(* Schneider Machine Expert - Basic project control, file version 2.9.0.0 *)
(* ProjectInformations: Name=Nuevo proyecto *)

HARDWARE
  Cpu 0: TM221M16R/G
  EthernetConfiguration: NetworkName=M221, IpAllocationMode=FixedAddress, IpAddress=0.0.0.0, SubnetMask=0.0.0.0
  SerialLineConfiguration: Baud=Baud19200, Parity=ParityEven, DataBits=DataBits8, StopBits=StopBits1, PhysicalMedium=PhysicalMediumRs485, TransmissionMode=TransmissionModeModbusRtu, SlaveId=1, Addressing=SlaveAddressing
  MastTask: UsePeriodScanMode=true, PeriodScan=50
  FastTask: Period=255
  CpuBehavior: StartingMode=StartAsPreviousState, AutoSaveRamOnEeprom=true, WatchdogPeriod=250

SYMBOLS  (address, symbol, comment, settings)
  %MW103    CONT
  %MW500    POSITION
  %MW501    VELOCITY
  %MW502    ANGLE
  %MW503    CRISP
  %MF1      POS_NL
  %MF3      POS_NM
  %MF5      POS_NP
  %MF7      POS_ZR
  %MF9      POS_PP
  %MF11     POS_PM
  %MF13     POS_PL
  %MF15     VEL_NL
  %MF17     VEL_NM
  %MF19     VEL_NP
  %MF21     VEL_ZR
  %MF23     VEL_PP
  %MF25     VEL_PM
  %MF27     VEL_PL
  %MF29     ANG_NL
  %MF31     ANG_NM
  %MF33     ANG_ZR
  %MF35     ANG_PM
  %MF37     ANG_PL
  %MF39     W10
  %MF41     W23
  %MF43     W24
  %MF45     W2
  %MF47     W5
  %MF49     W11
  %MF51     W15
  %MF53     W18
  %MF55     W21
  %MF57     W22
  %MF59     W3
  %MF61     W6
  %MF63     W12
  %MF65     W17
  %MF67     W20
  %MF69     W1
  %MF71     W4
  %MF73     W7
  %MF75     W8
  %MF77     W13
  %MF79     W16
  %MF81     W19
  %MF83     W9
  %MF85     W14
  %MF87     W25
  %MF89     NL
  %MF91     NM
  %MF93     ZR
  %MF95     PM
  %MF97     PL
  %MF99     NUM
  %MF101    DEN
  %KF1      MEAN_NL_POS  [Value=-3]
  %KF3      MEAN_NM_POS  [Value=-2]
  %KF5      MEAN_NP_POS  [Value=-1]
  %KF7      MEAN_ZR_POS  [Value=0]
  %KF9      MEAN_PP_POS  [Value=1]
  %KF11     MEAN_PM_POS  [Value=2]
  %KF13     MEAN_PL_POS  [Value=3]
  %KF15     SIGMA_POS  [Value=0.365]
  %KF17     MEAN_NL_VEL  [Value=-5]
  %KF19     MEAN_NM_VEL  [Value=-3.333]
  %KF21     MEAN_NP_VEL  [Value=-1.667]
  %KF23     MEAN_ZR_VEL  [Value=0]
  %KF25     MEAN_PP_VEL  [Value=1.667]
  %KF27     MEAN_PM_VEL  [Value=3.333]
  %KF29     MEAN_PL_VEL  [Value=5]
  %KF31     SIGMA_VEL  [Value=0.7]
  %KF33     MEAN_NL_THETA  [Value=-0.2618]
  %KF35     MEAN_NM_THETA  [Value=-0.1]
  %KF37     MEAN_ZR_THETA  [Value=0]
  %KF39     MEAN_PM_THETA  [Value=0.1]
  %KF41     MEAN_PL_THETA  [Value=0.2618]
  %KF43     SIGMA_L_THETA  [Value=0.085]
  %KF45     SIGMA_M_THETA  [Value=0.03]
  %KF47     SIGMA_Z_THETA  [Value=0.02]
  %KF49     MEAN_U_NL  [Value=-200]
  %KF51     MEAN_U_NM  [Value=-100]
  %KF53     MEAN_U_ZR  [Value=0]
  %KF55     MEAN_U_PM  [Value=100]
  %KF57     MEAN_U_PL  [Value=200]
  %KF59     SIGMA_L_U  [Value=50]
  %KF61     SIGMA_M_U  [Value=45]
  %KF63     SIGMA_Z_U  [Value=35]

POU Fuzzy
  (* SectionNumber=1 *)

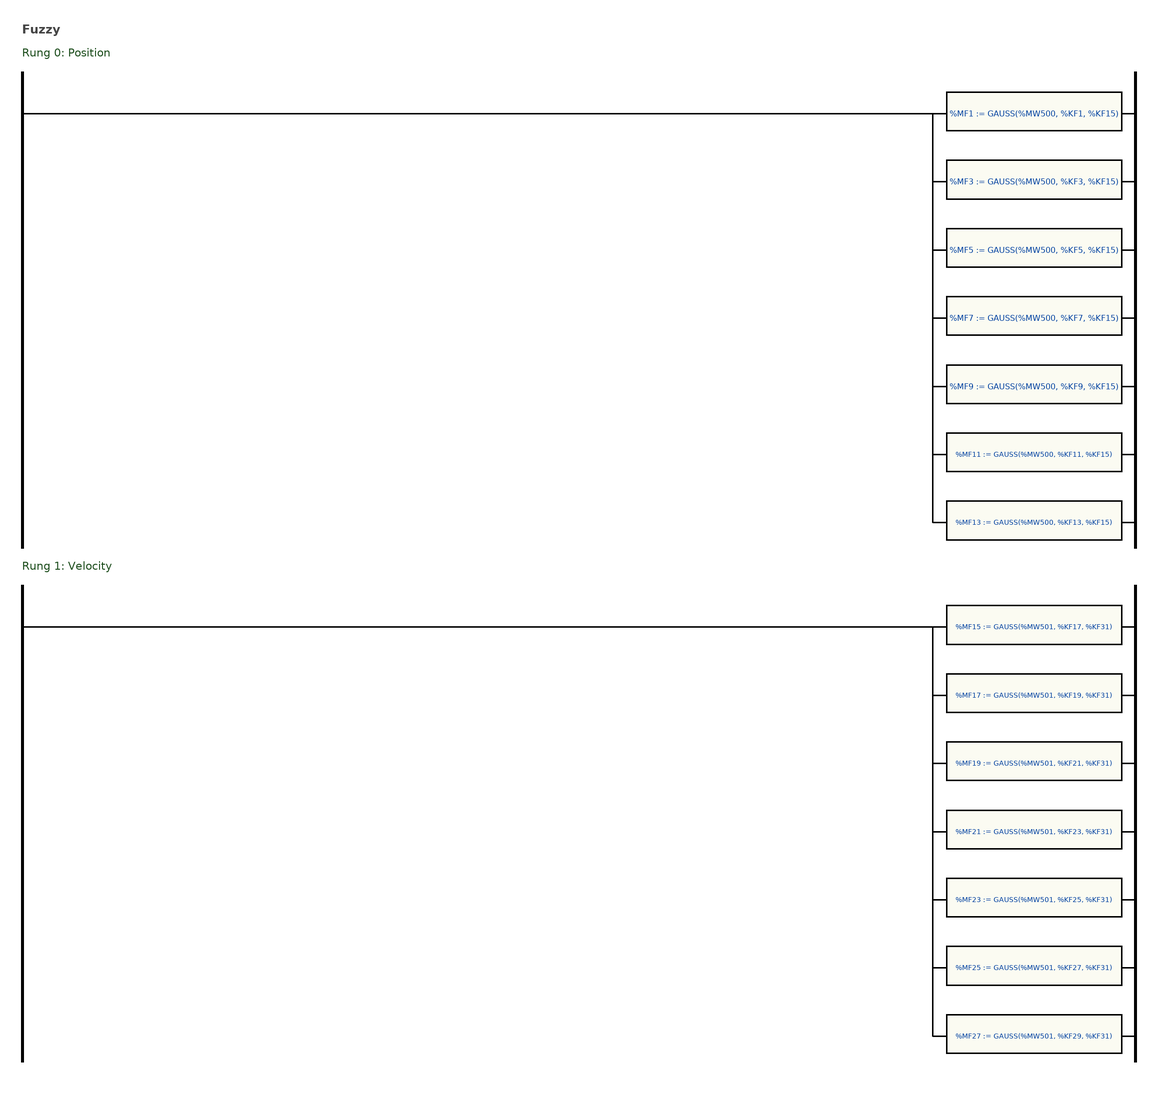

// Rung 0: Position
  LD 1
  [ %MF1 := GAUSS ( %MW500 , %KF1 , %KF15 ) ](* POS_NL, POSITION, MEAN_NL_POS, SIGMA_POS *)
  [ %MF3 := GAUSS ( %MW500 , %KF3 , %KF15 ) ](* POS_NM, POSITION, MEAN_NM_POS, SIGMA_POS *)
  [ %MF5 := GAUSS ( %MW500 , %KF5 , %KF15 ) ](* POS_NP, POSITION, MEAN_NP_POS, SIGMA_POS *)
  [ %MF7 := GAUSS ( %MW500 , %KF7 , %KF15 ) ](* POS_ZR, POSITION, MEAN_ZR_POS, SIGMA_POS *)
  [ %MF9 := GAUSS ( %MW500 , %KF9 , %KF15 ) ](* POS_PP, POSITION, MEAN_PP_POS, SIGMA_POS *)
  [ %MF11 := GAUSS ( %MW500 , %KF11 , %KF15 ) ](* POS_PM, POSITION, MEAN_PM_POS, SIGMA_POS *)
  [ %MF13 := GAUSS ( %MW500 , %KF13 , %KF15 ) ](* POS_PL, POSITION, MEAN_PL_POS, SIGMA_POS *)
  // as ST:
  //   POS_NL := GAUSS ( POSITION , MEAN_NL_POS , SIGMA_POS );
  //   POS_NM := GAUSS ( POSITION , MEAN_NM_POS , SIGMA_POS );
  //   POS_NP := GAUSS ( POSITION , MEAN_NP_POS , SIGMA_POS );
  //   POS_ZR := GAUSS ( POSITION , MEAN_ZR_POS , SIGMA_POS );
  //   POS_PP := GAUSS ( POSITION , MEAN_PP_POS , SIGMA_POS );
  //   POS_PM := GAUSS ( POSITION , MEAN_PM_POS , SIGMA_POS );
  //   POS_PL := GAUSS ( POSITION , MEAN_PL_POS , SIGMA_POS );

// Rung 1: Velocity
  LD 1
  [ %MF15 := GAUSS ( %MW501 , %KF17 , %KF31 ) ](* VEL_NL, VELOCITY, MEAN_NL_VEL, SIGMA_VEL *)
  [ %MF17 := GAUSS ( %MW501 , %KF19 , %KF31 ) ](* VEL_NM, VELOCITY, MEAN_NM_VEL, SIGMA_VEL *)
  [ %MF19 := GAUSS ( %MW501 , %KF21 , %KF31 ) ](* VEL_NP, VELOCITY, MEAN_NP_VEL, SIGMA_VEL *)
  [ %MF21 := GAUSS ( %MW501 , %KF23 , %KF31 ) ](* VEL_ZR, VELOCITY, MEAN_ZR_VEL, SIGMA_VEL *)
  [ %MF23 := GAUSS ( %MW501 , %KF25 , %KF31 ) ](* VEL_PP, VELOCITY, MEAN_PP_VEL, SIGMA_VEL *)
  [ %MF25 := GAUSS ( %MW501 , %KF27 , %KF31 ) ](* VEL_PM, VELOCITY, MEAN_PM_VEL, SIGMA_VEL *)
  [ %MF27 := GAUSS ( %MW501 , %KF29 , %KF31 ) ](* VEL_PL, VELOCITY, MEAN_PL_VEL, SIGMA_VEL *)
  // as ST:
  //   VEL_NL := GAUSS ( VELOCITY , MEAN_NL_VEL , SIGMA_VEL );
  //   VEL_NM := GAUSS ( VELOCITY , MEAN_NM_VEL , SIGMA_VEL );
  //   VEL_NP := GAUSS ( VELOCITY , MEAN_NP_VEL , SIGMA_VEL );
  //   VEL_ZR := GAUSS ( VELOCITY , MEAN_ZR_VEL , SIGMA_VEL );
  //   VEL_PP := GAUSS ( VELOCITY , MEAN_PP_VEL , SIGMA_VEL );
  //   VEL_PM := GAUSS ( VELOCITY , MEAN_PM_VEL , SIGMA_VEL );
  //   VEL_PL := GAUSS ( VELOCITY , MEAN_PL_VEL , SIGMA_VEL );

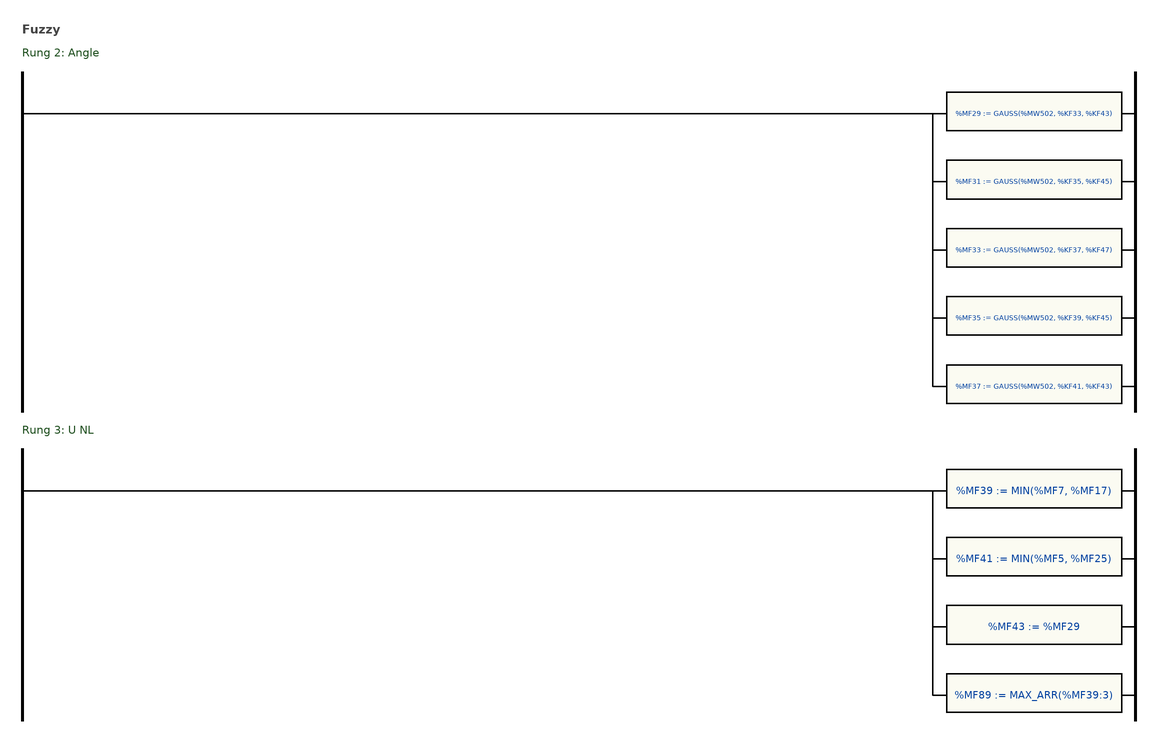

// Rung 2: Angle
  LD 1
  [ %MF29 := GAUSS ( %MW502 , %KF33 , %KF43 ) ](* ANG_NL, ANGLE, MEAN_NL_THETA, SIGMA_L_THETA *)
  [ %MF31 := GAUSS ( %MW502 , %KF35 , %KF45 ) ](* ANG_NM, ANGLE, MEAN_NM_THETA, SIGMA_M_THETA *)
  [ %MF33 := GAUSS ( %MW502 , %KF37 , %KF47 ) ](* ANG_ZR, ANGLE, MEAN_ZR_THETA, SIGMA_Z_THETA *)
  [ %MF35 := GAUSS ( %MW502 , %KF39 , %KF45 ) ](* ANG_PM, ANGLE, MEAN_PM_THETA, SIGMA_M_THETA *)
  [ %MF37 := GAUSS ( %MW502 , %KF41 , %KF43 ) ](* ANG_PL, ANGLE, MEAN_PL_THETA, SIGMA_L_THETA *)
  // as ST:
  //   ANG_NL := GAUSS ( ANGLE , MEAN_NL_THETA , SIGMA_L_THETA );
  //   ANG_NM := GAUSS ( ANGLE , MEAN_NM_THETA , SIGMA_M_THETA );
  //   ANG_ZR := GAUSS ( ANGLE , MEAN_ZR_THETA , SIGMA_Z_THETA );
  //   ANG_PM := GAUSS ( ANGLE , MEAN_PM_THETA , SIGMA_M_THETA );
  //   ANG_PL := GAUSS ( ANGLE , MEAN_PL_THETA , SIGMA_L_THETA );

// Rung 3: U NL
  LD 1
  [ %MF39 := MIN ( %MF7 , %MF17 ) ](* W10, POS_ZR, VEL_NM *)
  [ %MF41 := MIN ( %MF5 , %MF25 ) ](* W23, POS_NP, VEL_PM *)
  [ %MF43 := %MF29 ]      (* W24, ANG_NL *)
  [ %MF89 := MAX_ARR ( %MF39:3 ) ](* NL, W10 *)
  // as ST:
  //   W10 := MIN ( POS_ZR , VEL_NM );
  //   W23 := MIN ( POS_NP , VEL_PM );
  //   W24 := ANG_NL;
  //   NL := MAX_ARR ( W10:3 );

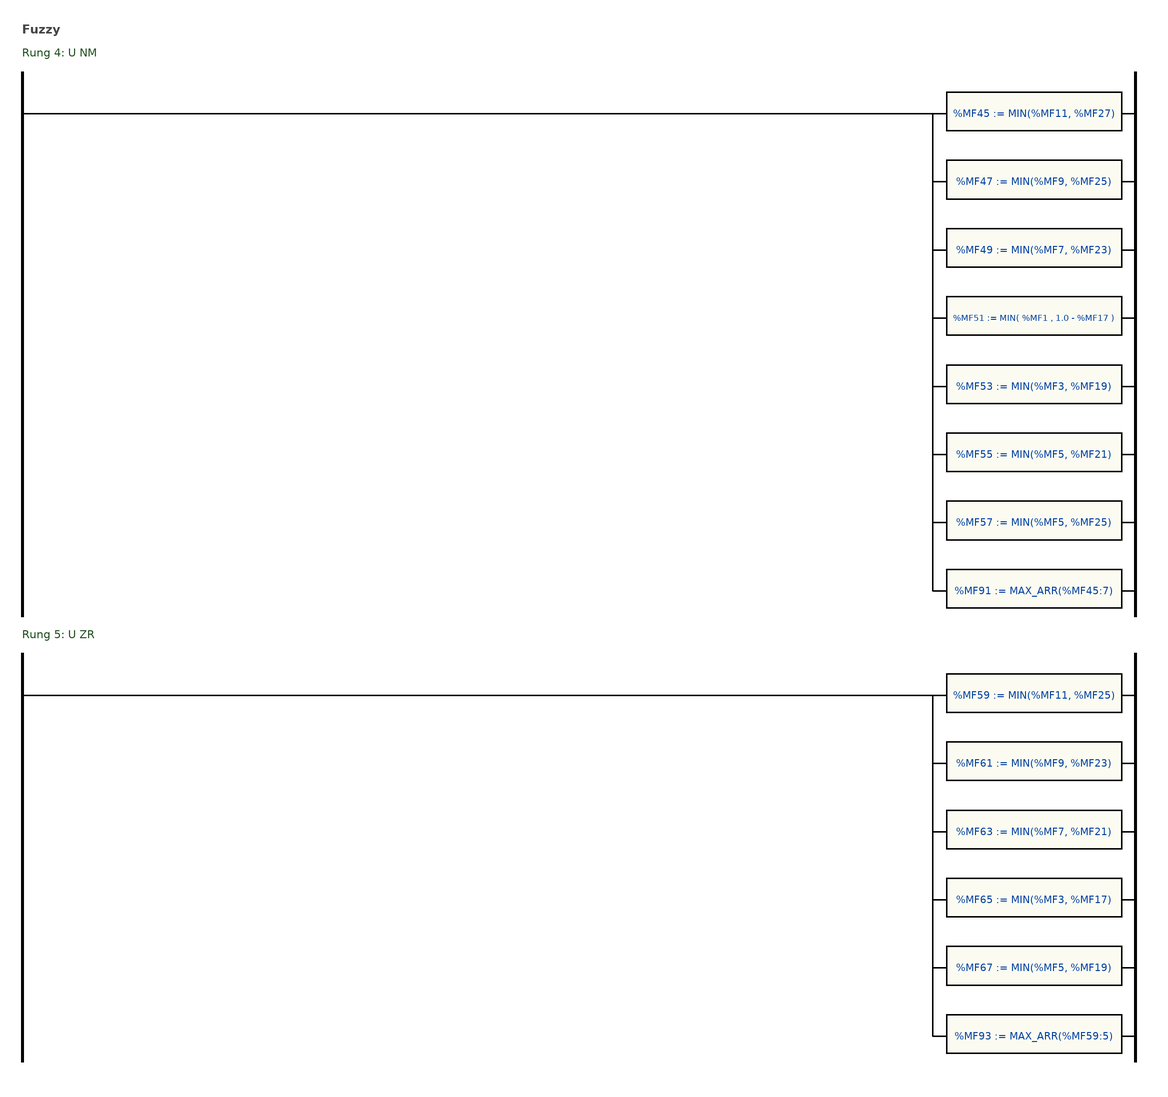

// Rung 4: U NM
  LD 1
  [ %MF45 := MIN ( %MF11 , %MF27 ) ](* W2, POS_PM, VEL_PL *)
  [ %MF47 := MIN ( %MF9 , %MF25 ) ](* W5, POS_PP, VEL_PM *)
  [ %MF49 := MIN ( %MF7 , %MF23 ) ](* W11, POS_ZR, VEL_PP *)
  [%MF51 := MIN( %MF1 , 1.0 - %MF17 )](* W15, POS_NL, VEL_NM *)
  [ %MF53 := MIN ( %MF3 , %MF19 ) ](* W18, POS_NM, VEL_NP *)
  [ %MF55 := MIN ( %MF5 , %MF21 ) ](* W21, POS_NP, VEL_ZR *)
  [ %MF57 := MIN ( %MF5 , %MF25 ) ](* W22, POS_NP, VEL_PM *)
  [ %MF91 := MAX_ARR ( %MF45:7 ) ](* NM, W2 *)
  // as ST:
  //   W2 := MIN ( POS_PM , VEL_PL );
  //   W5 := MIN ( POS_PP , VEL_PM );
  //   W11 := MIN ( POS_ZR , VEL_PP );
  //   W15 := MIN( POS_NL , 1.0 - VEL_NM );
  //   W18 := MIN ( POS_NM , VEL_NP );
  //   W21 := MIN ( POS_NP , VEL_ZR );
  //   W22 := MIN ( POS_NP , VEL_PM );
  //   NM := MAX_ARR ( W2:7 );

// Rung 5: U ZR
  LD 1
  [ %MF59 := MIN ( %MF11 , %MF25 ) ](* W3, POS_PM, VEL_PM *)
  [ %MF61 := MIN ( %MF9 , %MF23 ) ](* W6, POS_PP, VEL_PP *)
  [ %MF63 := MIN ( %MF7 , %MF21 ) ](* W12, POS_ZR, VEL_ZR *)
  [ %MF65 := MIN ( %MF3 , %MF17 ) ](* W17, POS_NM, VEL_NM *)
  [ %MF67 := MIN ( %MF5 , %MF19 ) ](* W20, POS_NP, VEL_NP *)
  [ %MF93 := MAX_ARR ( %MF59:5 ) ](* ZR, W3 *)
  // as ST:
  //   W3 := MIN ( POS_PM , VEL_PM );
  //   W6 := MIN ( POS_PP , VEL_PP );
  //   W12 := MIN ( POS_ZR , VEL_ZR );
  //   W17 := MIN ( POS_NM , VEL_NM );
  //   W20 := MIN ( POS_NP , VEL_NP );
  //   ZR := MAX_ARR ( W3:5 );

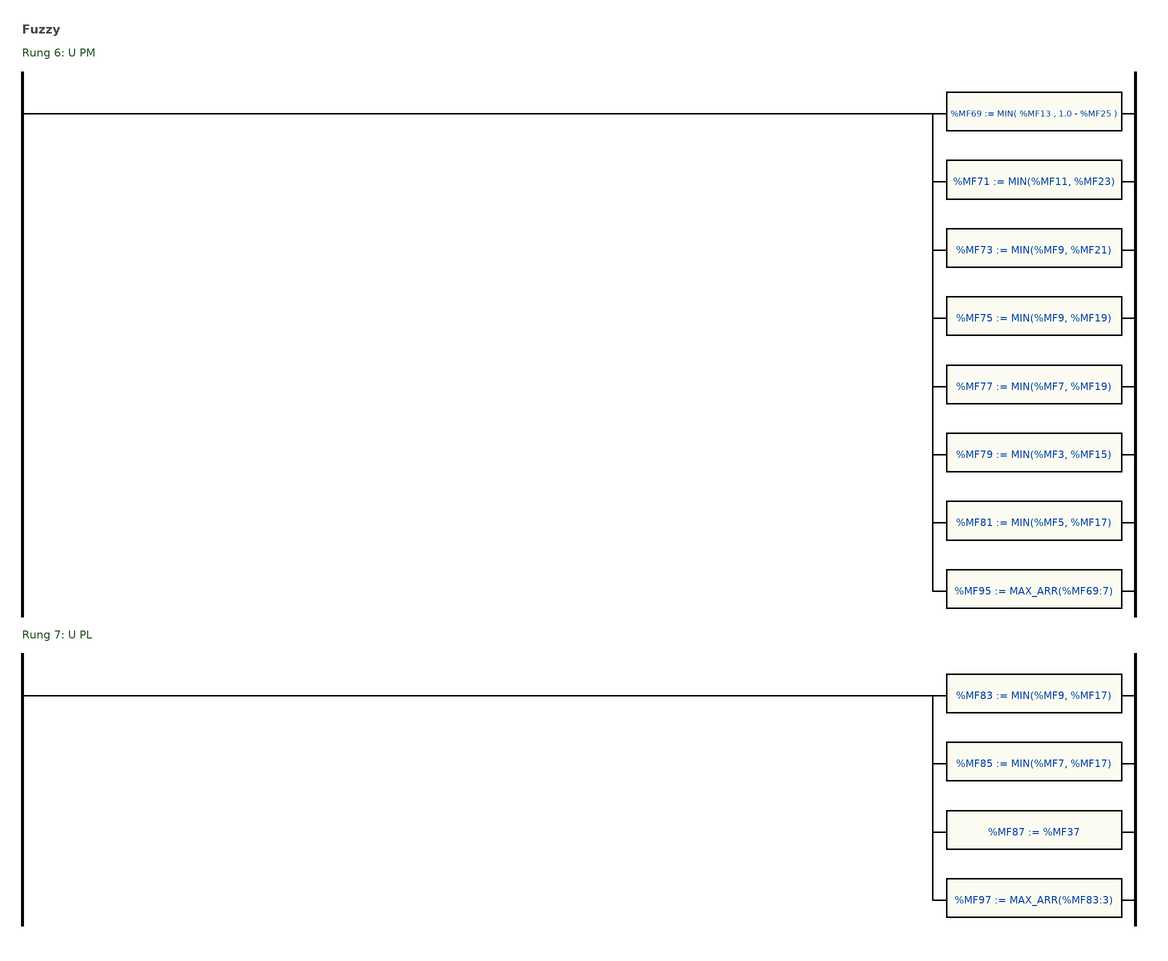

// Rung 6: U PM
  LD 1
  [%MF69 := MIN( %MF13 , 1.0 - %MF25 )](* W1, POS_PL, VEL_PM *)
  [ %MF71 := MIN ( %MF11 , %MF23 ) ](* W4, POS_PM, VEL_PP *)
  [ %MF73 := MIN ( %MF9 , %MF21 ) ](* W7, POS_PP, VEL_ZR *)
  [ %MF75 := MIN ( %MF9 , %MF19 ) ](* W8, POS_PP, VEL_NP *)
  [ %MF77 := MIN ( %MF7 , %MF19 ) ](* W13, POS_ZR, VEL_NP *)
  [ %MF79 := MIN ( %MF3 , %MF15 ) ](* W16, POS_NM, VEL_NL *)
  [ %MF81 := MIN ( %MF5 , %MF17 ) ](* W19, POS_NP, VEL_NM *)
  [ %MF95 := MAX_ARR ( %MF69:7 ) ](* PM, W1 *)
  // as ST:
  //   W1 := MIN( POS_PL , 1.0 - VEL_PM );
  //   W4 := MIN ( POS_PM , VEL_PP );
  //   W7 := MIN ( POS_PP , VEL_ZR );
  //   W8 := MIN ( POS_PP , VEL_NP );
  //   W13 := MIN ( POS_ZR , VEL_NP );
  //   W16 := MIN ( POS_NM , VEL_NL );
  //   W19 := MIN ( POS_NP , VEL_NM );
  //   PM := MAX_ARR ( W1:7 );

// Rung 7: U PL
  LD 1
  [ %MF83 := MIN ( %MF9 , %MF17 ) ](* W9, POS_PP, VEL_NM *)
  [ %MF85 := MIN ( %MF7 , %MF17 ) ](* W14, POS_ZR, VEL_NM *)
  [ %MF87 := %MF37 ]      (* W25, ANG_PL *)
  [ %MF97 := MAX_ARR ( %MF83:3 ) ](* PL, W9 *)
  // as ST:
  //   W9 := MIN ( POS_PP , VEL_NM );
  //   W14 := MIN ( POS_ZR , VEL_NM );
  //   W25 := ANG_PL;
  //   PL := MAX_ARR ( W9:3 );

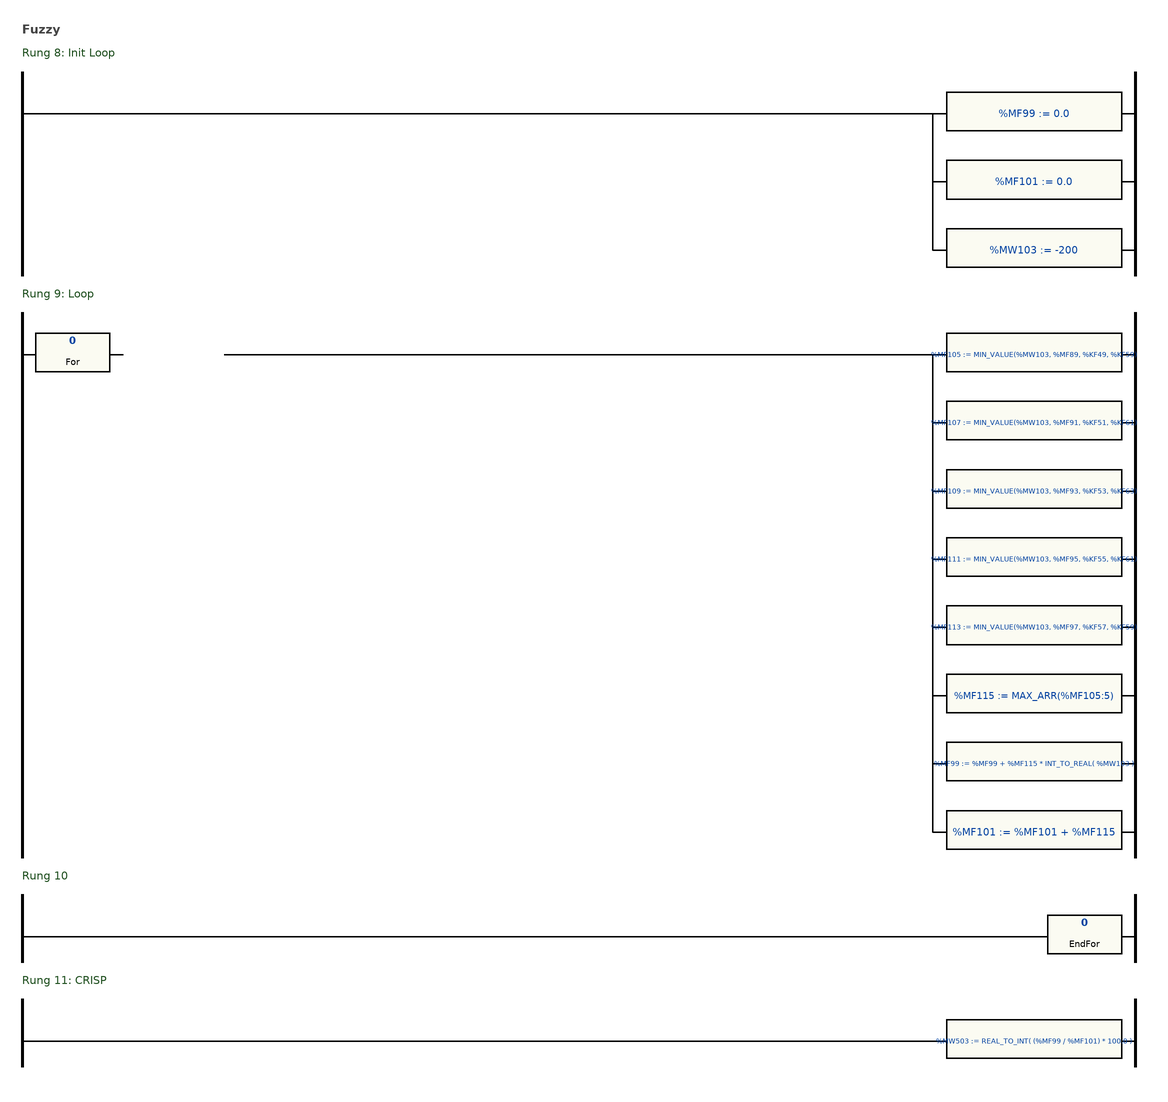

// Rung 8: Init Loop
  LD 1
  [ %MF99 := 0.0 ]        (* NUM *)
  [ %MF101 := 0.0 ]       (* DEN *)
  [ %MW103 := -200 ]      (* CONT *)
  // as ST:
  //   NUM := 0.0;
  //   DEN := 0.0;
  //   CONT := -200;

// Rung 9: Loop
  FOR0 ( %MW103, %MW103, <=, 200, 4 )(* CONT, CONT *)
  [ %MF105 := MIN_VALUE ( %MW103 , %MF89 , %KF49 , %KF59 ) ](* CONT, NL, MEAN_U_NL, SIGMA_L_U *)
  [ %MF107 := MIN_VALUE ( %MW103 , %MF91 , %KF51 , %KF61 ) ](* CONT, NM, MEAN_U_NM, SIGMA_M_U *)
  [ %MF109 := MIN_VALUE ( %MW103 , %MF93 , %KF53 , %KF63 ) ](* CONT, ZR, MEAN_U_ZR, SIGMA_Z_U *)
  [ %MF111 := MIN_VALUE ( %MW103 , %MF95 , %KF55 , %KF61 ) ](* CONT, PM, MEAN_U_PM, SIGMA_M_U *)
  [ %MF113 := MIN_VALUE ( %MW103 , %MF97 , %KF57 , %KF59 ) ](* CONT, PL, MEAN_U_PL, SIGMA_L_U *)
  [ %MF115 := MAX_ARR ( %MF105:5 ) ]
  [%MF99 := %MF99 + %MF115 * INT_TO_REAL( %MW103 )](* NUM, NUM, CONT *)
  [ %MF101 := %MF101 + %MF115 ](* DEN, DEN *)

// Rung 10
  LD 1
  ENDFOR0

// Rung 11: CRISP
  LD 1
  [%MW503 := REAL_TO_INT( (%MF99 / %MF101) * 100.0 )](* CRISP, NUM, DEN *)
  // as ST:
  //   CRISP := REAL_TO_INT( (NUM / DEN) * 100.0 );

UserFunctionPou GAUSS
  (* SectionNumber=2 *)

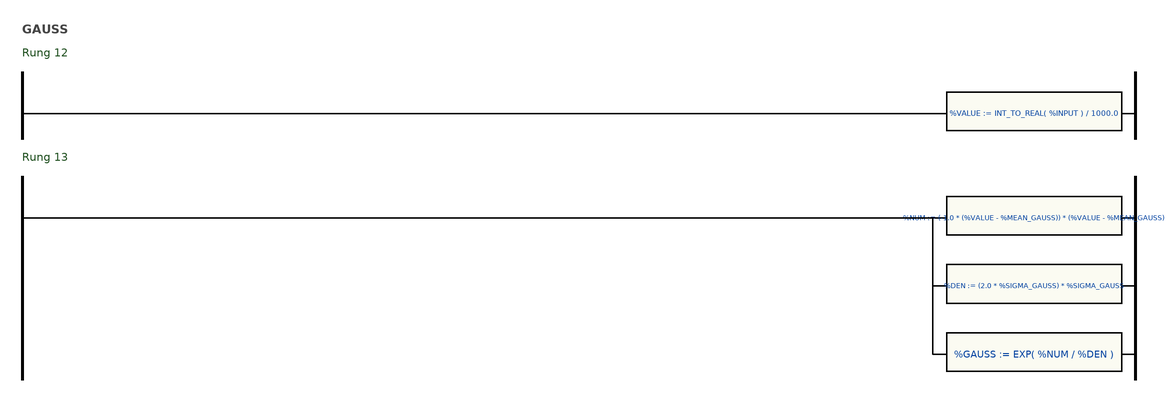

// Rung 12
  LD 1
  [%VALUE := INT_TO_REAL( %INPUT ) / 1000.0]
  // as ST:
  //   %VALUE := INT_TO_REAL( %INPUT ) / 1000.0;

// Rung 13
  LD 1
  [%NUM := (-1.0 * (%VALUE - %MEAN_GAUSS)) * (%VALUE - %MEAN_GAUSS)]
  [%DEN := (2.0 * %SIGMA_GAUSS) * %SIGMA_GAUSS]
  [%GAUSS := EXP( %NUM / %DEN )]
  // as ST:
  //   %NUM := (-1.0 * (%VALUE - %MEAN_GAUSS)) * (%VALUE - %MEAN_GAUSS);
  //   %DEN := (2.0 * %SIGMA_GAUSS) * %SIGMA_GAUSS;
  //   %GAUSS := EXP( %NUM / %DEN );

UserFunctionPou MIN
  (* SectionNumber=3 *)

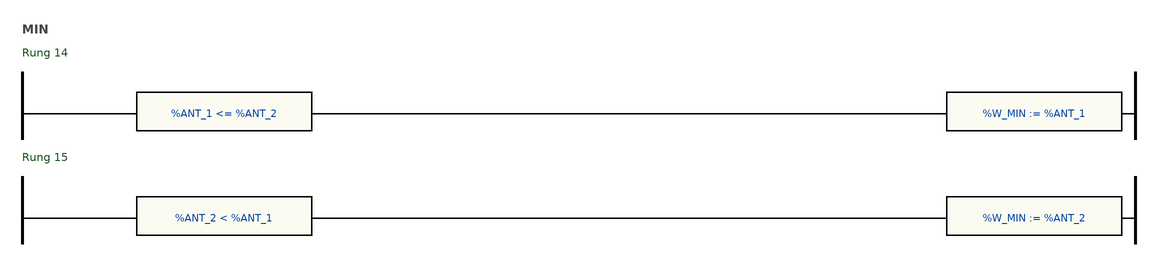

// Rung 14
  LD [%ANT_1 <= %ANT_2]
  [%W_MIN := %ANT_1]
  // as ST:
  //   IF %ANT_1 <= %ANT_2 THEN %W_MIN := %ANT_1; END_IF;

// Rung 15
  LD [%ANT_2 < %ANT_1]
  [%W_MIN := %ANT_2]
  // as ST:
  //   IF %ANT_2 < %ANT_1 THEN %W_MIN := %ANT_2; END_IF;

UserFunctionPou MIN_VALUE
  (* SectionNumber=4 *)

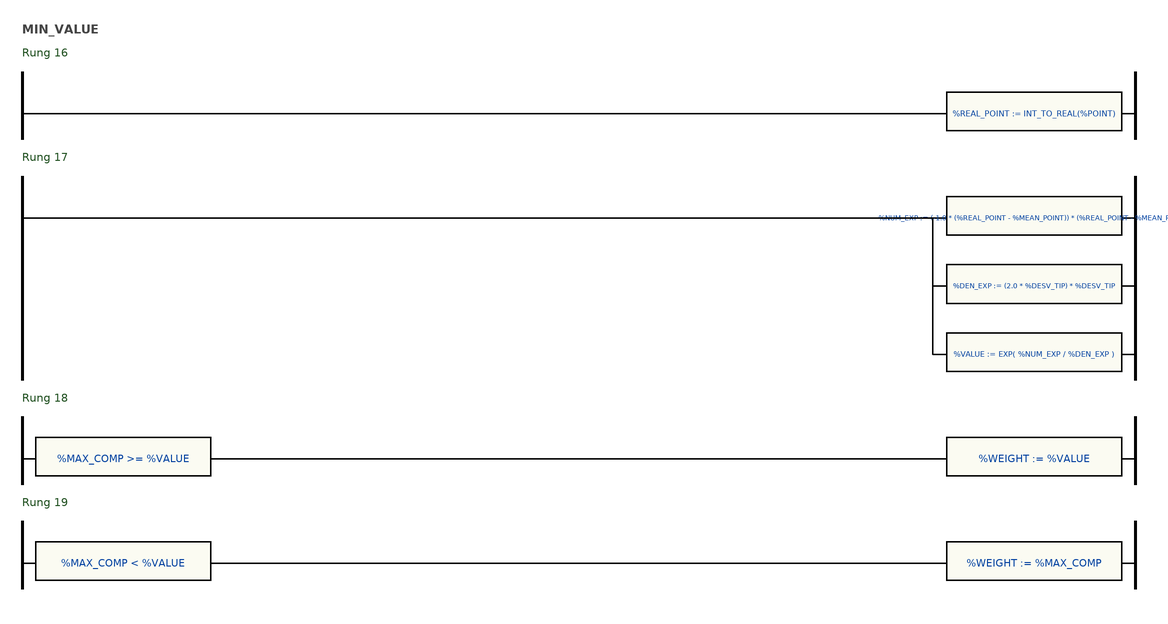

// Rung 16
  LD 1
  [%REAL_POINT := INT_TO_REAL(%POINT)]
  // as ST:
  //   %REAL_POINT := INT_TO_REAL(%POINT);

// Rung 17
  LD 1
  [%NUM_EXP := (-1.0 * (%REAL_POINT - %MEAN_POINT)) * (%REAL_POINT - %MEAN_POINT)]
  [%DEN_EXP := (2.0 * %DESV_TIP) * %DESV_TIP]
  [%VALUE := EXP( %NUM_EXP / %DEN_EXP )]
  // as ST:
  //   %NUM_EXP := (-1.0 * (%REAL_POINT - %MEAN_POINT)) * (%REAL_POINT - %MEAN_POINT);
  //   %DEN_EXP := (2.0 * %DESV_TIP) * %DESV_TIP;
  //   %VALUE := EXP( %NUM_EXP / %DEN_EXP );

// Rung 18
  LD [%MAX_COMP >= %VALUE]
  [%WEIGHT := %VALUE]
  // as ST:
  //   IF %MAX_COMP >= %VALUE THEN %WEIGHT := %VALUE; END_IF;

// Rung 19
  LD [%MAX_COMP < %VALUE]
  [%WEIGHT := %MAX_COMP]
  // as ST:
  //   IF %MAX_COMP < %VALUE THEN %WEIGHT := %MAX_COMP; END_IF;

UserFunctionPou MAX
  (* SectionNumber=5 *)

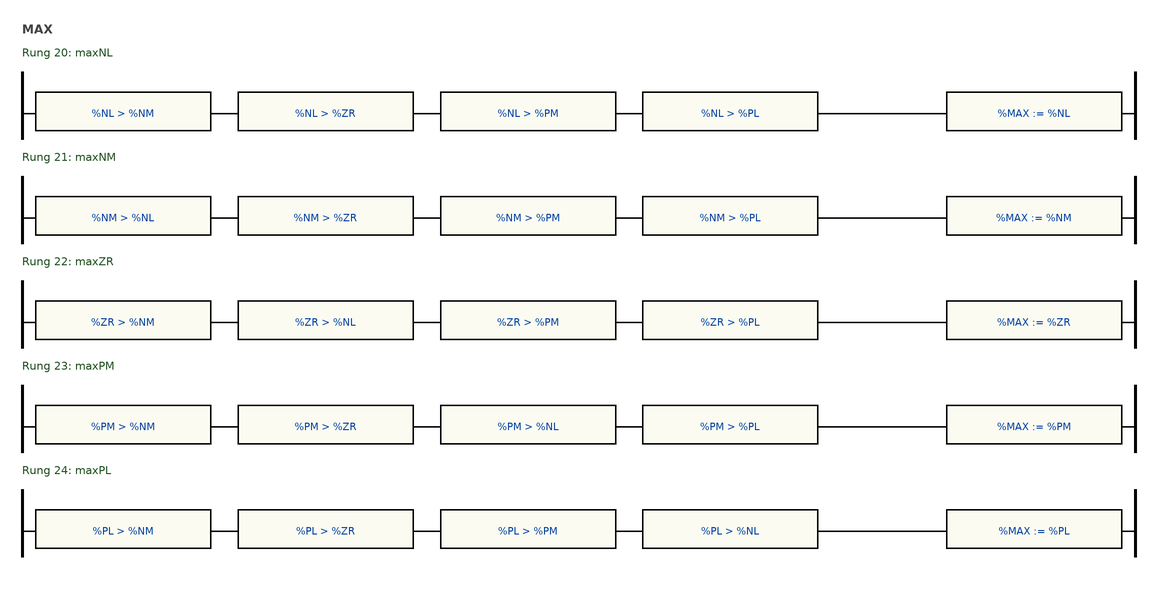

// Rung 20: maxNL
  LD [%NL > %NM]
  AND [%NL > %ZR]
  AND [%NL > %PM]
  AND [%NL > %PL]
  [%MAX := %NL]
  // as ST:
  //   IF %NL > %NM AND %NL > %ZR AND %NL > %PM AND %NL > %PL THEN %MAX := %NL; END_IF;

// Rung 21: maxNM
  LD [%NM > %NL]
  AND [%NM > %ZR]
  AND [%NM > %PM]
  AND [%NM > %PL]
  [%MAX := %NM]
  // as ST:
  //   IF %NM > %NL AND %NM > %ZR AND %NM > %PM AND %NM > %PL THEN %MAX := %NM; END_IF;

// Rung 22: maxZR
  LD [%ZR > %NM]
  AND [%ZR > %NL]
  AND [%ZR > %PM]
  AND [%ZR > %PL]
  [%MAX := %ZR]
  // as ST:
  //   IF %ZR > %NM AND %ZR > %NL AND %ZR > %PM AND %ZR > %PL THEN %MAX := %ZR; END_IF;

// Rung 23: maxPM
  LD [%PM > %NM]
  AND [%PM > %ZR]
  AND [%PM > %NL]
  AND [%PM > %PL]
  [%MAX := %PM]
  // as ST:
  //   IF %PM > %NM AND %PM > %ZR AND %PM > %NL AND %PM > %PL THEN %MAX := %PM; END_IF;

// Rung 24: maxPL
  LD [%PL > %NM]
  AND [%PL > %ZR]
  AND [%PL > %PM]
  AND [%PL > %NL]
  [%MAX := %PL]
  // as ST:
  //   IF %PL > %NM AND %PL > %ZR AND %PL > %PM AND %PL > %NL THEN %MAX := %PL; END_IF;
